// TwinCAT 3 PLC project PLC1
// ProgramVersion: 3.1.4020.5
// libraries:
//   Tc2_ModbusRTU, * (Beckhoff Automation GmbH)
//   Tc2_SerialCom, * (Beckhoff Automation GmbH)
//   Tc2_Standard, * (Beckhoff Automation GmbH)
//   Tc2_System, * (Beckhoff Automation GmbH)
//   Tc3_Module, * (Beckhoff Automation GmbH)
// project tree:
//   DUTs/SH200A/ ST_LoggedValues.TcDUT, ST_Simplex_Halt.TcDUT, ST_Simplex_Jog.TcDUT, ST_Simplex_Reset.TcDUT, ST_Simplex_SetPosition.TcDUT, ST_Simplex_Stop.TcDUT
//   / PlcTask.TcTTO
//   POUs/ FB_Simplex.TcPOU, MAIN.TcPOU
//   POUs/ModbusRTU/ ModbusRTU.TcGVL, SerialCommunication.TcPOU
// real-time tasks:
//   TASK PlcTask: cycle T#2ms, priority 20, ADS port 350
// I/O:
//   DEVICE Device 1 (EtherCAT), AmsNetId 192.168.1.100.2.1
//     Term 1 (EK1200) [EK1200-5000 EtherCAT Power supply (2A E-Bus)]
//       Term 2 (EL1008) [EL1008 8Ch. Dig. Input 24V, 3ms]
//       Term 3 (EL2008) [EL2008 8Ch. Dig. Output 24V, 0.5A]
//       Term 4 (EL9510) [EL9510 Power supply terminal 10V]
//       Term 5 (EL3356) [EL3356 1Ch. Ana. Input Resistor Bridge Terminal, 16bit, High Precision]
//       Term 6 (EL9011) [EL9011 End Terminal]
//   DEVICE Device 3 (EtherCAT), AmsNetId 192.168.1.100.4.1
//     Term 7 (EP6002-0002) [EP6002-0002 Interface (RS232/422/485)]
//   DEVICE Device 2 (COM Port)
// variable links:
//   PLC1/PLC1 Instance <-> Device 3 (EtherCAT)/Term 7 (EP6002-0002)
//     PlcTask Inputs/MAIN.fbSH200A.fbModbusRTUMaster.InData/D <-> COM TxPDO-Map Inputs Channel 1/Data In 0
//     PlcTask Inputs/MAIN.fbSH200A.fbModbusRTUMaster.InData/D @bit {8..168 step 8} <-> COM TxPDO-Map Inputs Channel 1/Data In {1..21}  (21 links)
//     PlcTask Inputs/MAIN.fbSH200A.fbModbusRTUMaster.InData/Status <-> COM TxPDO-Map Inputs Channel 1/Status
//     PlcTask Outputs/MAIN.fbSH200A.fbModbusRTUMaster.OutData/Ctrl <-> COM RxPDO-Map Outputs Channel 1/Ctrl
//     PlcTask Outputs/MAIN.fbSH200A.fbModbusRTUMaster.OutData/D <-> COM RxPDO-Map Outputs Channel 1/Data Out 0
//     PlcTask Outputs/MAIN.fbSH200A.fbModbusRTUMaster.OutData/D @bit {8..168 step 8} <-> COM RxPDO-Map Outputs Channel 1/Data Out {1..21}  (21 links)

CONFIGURATION PLC1
    RESOURCE PLC ON TwinCAT3
        TASK PlcTask(INTERVAL := T#2ms, PRIORITY := 20);
        PROGRAM MAIN WITH PlcTask : MAIN;
    END_RESOURCE
END_CONFIGURATION

// ---- DUTs/SH200A/ST_LoggedValues.TcDUT
TYPE ST_LoggedValues :
STRUCT
	nMotorFluxVoltage : INT;
END_STRUCT
END_TYPE

// ---- DUTs/SH200A/ST_Simplex_Halt.TcDUT
TYPE ST_Simplex_Halt :
STRUCT
	nMotorFluxVoltage : INT;
END_STRUCT
END_TYPE

// ---- DUTs/SH200A/ST_Simplex_Jog.TcDUT
TYPE ST_Simplex_Jog :
STRUCT
	fbTimerWriteModbus		: TON;		// Timer for writing values to Modbus
	bWriteControlOption		: BOOL;		// First state, define control mode
		nControlSetting		: UINT := 21; // Default value is set to position ramp control
	bWriteSetpointSpeed		: BOOL; 	// Second state, define maximum speed
		nMaxVelocity		: INT; 		// Maximum allowed velocity
		bSettingsDone		: BOOL;
	bJogForward				: BOOL;		// Third state, jogging forwards
	bJogBackwards			: BOOL;		// Fourth state, jogging backwards
		fbTimerWritePosition : TON;
		bSendPosition_MSB	: BOOL; // New setpoint sent to the motor Register! 
		bSendPosition_LSB	: BOOL; // New setpoint sent to the motor Register!
		bReadPosition		: BOOL;	// State inside jogg (all data is sent) 
	dnPosition				: DINT; // Current position of the motor
	
	//fAcceleration:LREAL;
	//fDeceleration:LREAL;
	//fJerk:LREAL;
	bDone	: BOOL;
	bBusy	: BOOL;
	bActive	: BOOL;
	bCommandAborted	: BOOL;
	bError	 : BOOL;
	nErrorID : UDINT;
END_STRUCT
END_TYPE

// ---- DUTs/SH200A/ST_Simplex_Reset.TcDUT
TYPE ST_Simplex_Reset :
STRUCT
END_STRUCT
END_TYPE

// ---- DUTs/SH200A/ST_Simplex_SetPosition.TcDUT
TYPE ST_Simplex_SetPosition :
STRUCT
	bExecute:BOOL;
	fPosition:LREAL;
	bMode:BOOL;
	//	stOptions:ST_SetPositionOptions;
	bDone:BOOL;
	bBusy:BOOL;
	bError:BOOL;
	nErrorID:UDINT;
END_STRUCT
END_TYPE

// ---- DUTs/SH200A/ST_Simplex_Stop.TcDUT
TYPE ST_Simplex_Stop :
STRUCT
	bExecute:BOOL;
	fDeceleration:LREAL;
	fJerk:LREAL;
	//stOptions:ST_MoveOptions;
	bDone:BOOL;
	bBusy:BOOL;
	bActive:BOOL;
	bCommandAborted:BOOL;
	bError:BOOL;
	nErrorID:UDINT;
END_STRUCT
END_TYPE

// ---- POUs/ModbusRTU/ModbusRTU.TcGVL
VAR_GLOBAL
	COMin_EL60XX AT %I* : KL6InData22B;
	COMout_EL60XX AT %Q* : KL6OutData22B;
	RxBuffer: Combuffer;
	TxBuffer: Combuffer;
END_VAR

// ---- POUs/MAIN.TcPOU
PROGRAM MAIN
VAR
	fbSH200A : FB_Simplex();
END_VAR

fbSH200A.M_Jog();
//fbSH200A.M_LogValues();
SerialCommunication();
//fbSH200A();

END_PROGRAM

// ---- POUs/FB_Simplex.TcPOU
FUNCTION_BLOCK FB_Simplex
VAR
	(* Stored Motor Parameters *)
	bWriteData	: BOOL;

	nTorqueLimit		: INT  := 3; // TorqueLimit for the motor  
	rM_SetPointSpeed	: REAL := 10;		 // Setpoint from user (cmm/s) 
	unControlOption		: UINT := 32;
	
	dnCenterPosition	: DINT;
	dnCCVEndPosition	: DINT := -200000;
	dnCVEndPosition		: DINT := 200000;

	dnPosRegMSB			: DINT;
	dnPosRegLSB			: DINT;
	
	fbModbusRTUMaster 	: MODbusRtuMaster_KL6x22B;
		unVersionNumber		: UINT;
		bMBAddress			: BYTE;
		unQuantity			: UINT; 
		unMBAddr			: UINT;
		unDataLength		: UINT;
		bStartReading		: BOOL;
		unTimeOut			: TIME := T#5S;	
		bBusy				: BOOL;
		bError				: BOOL;
		unErrorID			: UINT;
		unReadBytes			: UINT;
		lnPosition			: LINT;
		SPosition			: DINT;
		nCurr				: INT; // Read register 223	
	stSimplex_SetPosition	: ST_Simplex_SetPosition();	
	stSimplex_Jog			: ST_Simplex_Jog();
	stSimplex_Stop			: ST_Simplex_Stop();
	stSimplex_Reset			: ST_Simplex_Reset();
	stSimplex_Halt			: ST_Simplex_Halt();
	stLoggedValues			: ST_LoggedValues();
	dnRedMSB: BYTE;
END_VAR

(*		fbModbusRTUMaster(	UnitID   := 1,
						  	Quantity := 2,
							MBAddr	 := 200,
							cbLength := 4,
							pMemoryAddr := ADR(lnPosition),
							Execute		:= bWriteData, 
							TimeOut		:= T#5S, 
							Busy		=> bBusy, 
							Error		=> bError,
							ErrorId		=> unErrorID,
							cbRead		=> unReadBytes);		
		fbModbusRTUMaster.ReadRegs();
 *)
 (*
 	fbModbusRTUMaster(	UnitID   := 1,
					  	Quantity := 1,
						MBAddr	 := 449,
						cbLength := 16,
						pMemoryAddr := ADR(dnPosRegMsb),
						Execute		:= bWriteData, 
						TimeOut		:= T#5S, 
						Busy		=> bBusy, 
						Error		=> bError,
						ErrorId		=> unErrorID,
						cbRead		=> unReadBytes);		
	fbModbusRTUMaster.WriteRegs();
*)

{warning 'add method implementation'}
METHOD M_checkNC_settings : BOOL
VAR_INPUT
	//AXIS_REF	: REFERENCE TO Tc2_MC2.AXIS_REF;
END_VAR
END_METHOD

METHOD M_Jog : BOOL
VAR_INPUT
END_VAR
VAR
	bWrite 	: BOOL;	// Write command to Simplex motor
END_VAR
IF stSimplex_Jog.bActive THEN
	stSimplex_Jog.bWriteControlOption := TRUE;
	stSimplex_Jog.bActive := FALSE;
	stSimplex_Jog.bBusy := TRUE;
END_IF

// State to send setpoint velocity to SH200A
IF stSimplex_Jog.bWriteControlOption THEN
	stSimplex_Jog.fbTimerWriteModbus(PT := T#200MS);
	stSimplex_Jog.fbTimerWriteModbus(IN := TRUE);
	IF stSimplex_Jog.fbTimerWriteModbus.Q THEN
		bWrite := TRUE;
		fbModbusRTUMaster(	UnitID   := 1,
						  	Quantity := 1,
							MBAddr	 := 399,
							cbLength := 2,
							pMemoryAddr := ADR(stSimplex_Jog.nControlSetting),
							Execute		:= bWrite, 
							TimeOut		:= T#5S, 
							Busy		=> bBusy, 
							Error		=> bError,
							ErrorId		=> unErrorID,
							cbRead		=> unReadBytes);		
		stSimplex_Jog.bWriteControlOption := FALSE; 
		stSimplex_Jog.bWriteSetPointSpeed := TRUE;
		stSimplex_Jog.fbTimerWriteModbus(IN := FALSE);
	ELSE
		bWrite := FALSE;
		fbModbusRTUMaster(Execute := FALSE);
	END_IF	
	fbModbusRTUMaster.WriteSingleRegister();
	

// State to send control option to SH200A
ELSIF stSimplex_Jog.bWriteSetpointSpeed THEN 
	IF stSimplex_Jog.bSettingsDone THEN
		stSimplex_Jog.bJogForward 			:= TRUE;
		stSimplex_Jog.bSendPosition_LSB 	:= TRUE; 
		stSimplex_Jog.bSendPosition_MSB 	:= TRUE; 
		stSimplex_Jog.bWriteSetPointSpeed 	:= FALSE;
		stSimplex_Jog.bSettingsDone			:= FALSE;
	END_IF
		
	stSimplex_Jog.fbTimerWriteModbus(PT := T#200MS);
	stSimplex_Jog.fbTimerWriteModbus(IN := TRUE);
	stSimplex_Jog.nMaxVelocity := M_MM_TO_SPEED(rMM_SetPoint := rM_SetPointSpeed);
	
	IF stSimplex_Jog.fbTimerWriteModbus.Q THEN
		bWrite := TRUE;
		fbModbusRTUMaster( UnitID   	:= 1,
						   quantity 	:= 1,
						   MBAddr	 	:= 350,
						   cbLength 	:= 2,
						   pMemoryAddr 	:= ADR(stSimplex_Jog.nMaxVelocity),
						   Execute		:= bWrite, 
						   TimeOut		:= T#5S, 
						   Busy			=> bBusy, 
						   Error		=> bError,
						   ErrorId		=> unErrorID,
						   cbRead		=> unReadBytes);	
		stSimplex_Jog.fbTimerWriteModbus(IN := FALSE);
		stSimplex_Jog.bSettingsDone := TRUE;
	ELSE
		bWrite := FALSE;
		fbModbusRTUMaster(Execute := FALSE);
	END_IF
	fbModbusRTUMaster.WriteSingleRegister();
(* STATE 3: JOGGING FORWARD*)
ELSIF stSimplex_Jog.bJogForward THEN
	// Data formatting for Modbus (protcol is broken in the motor)
	dnPosRegMSB := (dnCVEndPosition AND 2#11111111111111110000000000000000);
	dnPosRegLSB := (dnCVEndPosition AND 2#00000000000000001111111111111111);
	
	// If we are done with set-up of new set point read the position for the motor
	IF stSimplex_Jog.bReadPosition THEN
		// Read position from motor
		bWrite := TRUE;
		fbModbusRTUMaster( 	UnitID   	:= 1,
					  		Quantity 	:= 2,
					   		MBAddr	 	:= 200,
					   		cbLength 	:= 4,
					   		pMemoryAddr := ADR(stSimplex_Jog.dnPosition),
					   		Execute		:= bWrite, 
					   		TimeOut		:= T#5S, 
					   		Busy		=> bBusy, 
					   		Error		=> bError,
					   		ErrorId		=> unErrorID,
					   		cbRead		=> unReadBytes);		
		stSimplex_Jog.fbTimerWriteModbus(IN := FALSE);
		fbModbusRTUMaster.ReadRegs();
		IF NOT(bBusy) AND unReadBytes <> 0 THEN
			bWrite := FALSE;
			fbModbusRTUMaster.Execute := FALSE;
		END_IF
	END_IF
	
	IF stSimplex_Jog.bSendPosition_LSB AND stSimplex_Jog.bSendPosition_MSB THEN
		stSimplex_Jog.fbTimerWriteModbus(PT := T#10MS);
		stSimplex_Jog.fbTimerWriteModbus(IN := TRUE);
		
		IF stSimplex_Jog.fbTimerWriteModbus.Q THEN
			fbModbusRTUMaster(	UnitID   := 1,
								Quantity := 1,
								MBAddr	 := 449,
								cbLength := 16,
								pMemoryAddr := ADR(dnPosRegMSB),
								Execute		:= bWrite, 
								TimeOut		:= T#5S, 
								Busy		=> bBusy, 
								Error		=> bError,
								ErrorId		=> unErrorID,
								cbRead		=> unReadBytes);		
			fbModbusRTUMaster.WriteRegs();
			StSimplex_Jog.bSendPosition_MSB := FALSE;
			stSimplex_Jog.fbTimerWriteModbus(IN := FALSE);
		ELSE
			bWrite := FALSE;
			fbModbusRTUMaster(Execute := FALSE);
		END_IF
	ELSIF NOT(stSimplex_Jog.bSendPosition_MSB) AND stSimplex_Jog.bSendPosition_LSB THEN
		stSimplex_Jog.fbTimerWriteModbus(PT := T#10MS);
		stSimplex_Jog.fbTimerWriteModbus(IN := TRUE);
		
		IF stSimplex_Jog.fbTimerWriteModbus.Q THEN
			bWrite := TRUE;
			fbModbusRTUMaster(	UnitID   := 1,
								Quantity := 1,
								MBAddr	 := 450,
								cbLength := 16,
								pMemoryAddr := ADR(dnPosRegLSB),
								Execute		:= bWrite, 
								TimeOut		:= T#5S, 
								Busy		=> bBusy, 
								Error		=> bError,
								ErrorId		=> unErrorID,
								cbRead		=> unReadBytes);		
			fbModbusRTUMaster.WriteRegs();
			StSimplex_Jog.bSendPosition_LSB := FALSE;	
			stSimplex_Jog.fbTimerWriteModbus(IN := FALSE);
		ELSE
			bWrite := FALSE;
			fbModbusRTUMaster(Execute := FALSE);
		END_IF
	ELSIF NOT(stSimplex_Jog.bSendPosition_MSB) AND NOT(stSimplex_Jog.bSendPosition_LSB) THEN
		fbModbusRTUMaster.WriteRegs();
		stSimplex_Jog.bReadPosition := TRUE;
	END_IF		

	IF stSimplex_Jog.dnPosition >= dnCVEndPosition THEN
		stSimplex_Jog.bJogForward		:= FALSE;
		stSimplex_Jog.bJogBackwards 	:= TRUE;
		stSimplex_Jog.bReadPosition 	:= FALSE;
		stSimplex_Jog.bSendPosition_LSB := TRUE;
		stSimplex_Jog.bSendPosition_MSB := TRUE;
		fbModbusRTUMaster.Execute 		:= FALSE;
	END_IF

(* STATE 4: JOGGING BACKWARDS*)
ELSIF stSimplex_Jog.bJogBackwards THEN
	dnPosRegMSB := (dnCCVEndPosition AND 2#11111111111111110000000000000000);
	dnPosRegLSB := (dnCCVEndPosition AND 2#00000000000000001111111111111111);
	
	// Read the position of the motor (True if we are done with the set-up)
	IF stSimplex_Jog.bReadPosition THEN
		// Read position from motor
		bWrite := TRUE;
		fbModbusRTUMaster( 	UnitID   	:= 1,
					  		Quantity 	:= 2,
					   		MBAddr	 	:= 200,
					   		cbLength 	:= 4,
					   		pMemoryAddr := ADR(stSimplex_Jog.dnPosition),
					   		Execute		:= bWrite, 
					   		TimeOut		:= T#5S, 
					   		Busy		=> bBusy, 
					   		Error		=> bError,
					   		ErrorId		=> unErrorID,
					   		cbRead		=> unReadBytes);		
		fbModbusRTUMaster.ReadRegs();
		IF NOT(bBusy) AND unReadBytes <> 0 THEN
			bWrite := FALSE;
			fbModbusRTUMaster.Execute := FALSE;
		END_IF
	END_IF		
	
	IF stSimplex_Jog.bSendPosition_LSB AND stSimplex_Jog.bSendPosition_MSB THEN
		stSimplex_Jog.fbTimerWriteModbus(PT := T#10MS);
		stSimplex_Jog.fbTimerWriteModbus(IN := TRUE);
		
		IF stSimplex_Jog.fbTimerWriteModbus.Q THEN
			fbModbusRTUMaster(	UnitID   := 1,
								Quantity := 1,
								MBAddr	 := 449,
								cbLength := 16,
								pMemoryAddr := ADR(dnPosRegMSB),
								Execute		:= bWrite, 
								TimeOut		:= T#5S, 
								Busy		=> bBusy, 
								Error		=> bError,
								ErrorId		=> unErrorID,
								cbRead		=> unReadBytes);
			stSimplex_Jog.fbTimerWriteModbus(IN := FALSE);
			fbModbusRTUMaster.WriteRegs();
			StSimplex_Jog.bSendPosition_MSB := FALSE;
		ELSE
			bWrite := FALSE;
			fbModbusRTUMaster(Execute := FALSE);
		END_IF
	ELSIF NOT(stSimplex_Jog.bSendPosition_MSB) AND stSimplex_Jog.bSendPosition_LSB THEN	
		stSimplex_Jog.fbTimerWriteModbus(PT := T#10MS);
		stSimplex_Jog.fbTimerWriteModbus(IN := TRUE);
		
		IF stSimplex_Jog.fbTimerWriteModbus.Q THEN
			bWrite := TRUE;
			fbModbusRTUMaster(	UnitID   := 1,
								Quantity := 1,
								MBAddr	 := 450,
								cbLength := 16,
								pMemoryAddr := ADR(dnPosRegLSB),
								Execute		:= bWrite, 
								TimeOut		:= T#5S, 
								Busy		=> bBusy, 
								Error		=> bError,
								ErrorId		=> unErrorID,
								cbRead		=> unReadBytes);
			stSimplex_Jog.fbTimerWriteModbus(IN := FALSE);		
			fbModbusRTUMaster.WriteRegs();
			StSimplex_Jog.bSendPosition_LSB := FALSE;	
		ELSE
			bWrite := FALSE;
			fbModbusRTUMaster(Execute := FALSE);
		END_IF
	ELSIF NOT(stSimplex_Jog.bSendPosition_MSB) AND NOT(stSimplex_Jog.bSendPosition_LSB) THEN
		fbModbusRTUMaster.WriteRegs();
		stSimplex_Jog.bReadPosition := TRUE;
	END_IF
	
	IF stSimplex_Jog.dnPosition >= dnCCVEndPosition THEN
		stSimplex_Jog.bJogForward		:= TRUE;
		stSimplex_Jog.bJogBackwards 	:= FALSE;
		stSimplex_Jog.bReadPosition 	:= FALSE;
		stSimplex_Jog.bSendPosition_LSB := TRUE;
		stSimplex_Jog.bSendPosition_MSB := TRUE;
		fbModbusRTUMaster.Execute 		:= FALSE;
	END_IF	
END_IF

IF stSimplex_Jog.bDone OR stSimplex_Jog.bCommandAborted THEN
	stSimplex_Jog.bJogForward			:= FALSE;
	stSimplex_Jog.bJogBackwards 		:= FALSE;
	stSimplex_Jog.bWriteSetpointSpeed 	:= FALSE;
	stSimplex_Jog.bWriteControlOption 	:= FALSE;
	stSimplex_Jog.bBusy   				:= FALSE;
	stSimplex_Jog.bActive 				:= FALSE;
END_IF
END_METHOD

METHOD M_LogValues : BOOL
VAR_INPUT
	//AXIS_REF	: REFERENCE TO Tc2_MC2.AXIS_REF;
END_VAR
VAR
	nValue : INT;
	nReadBytes : UINT;
END_VAR
(*
IF NOT(bBusy) THEN
	fbModbusRTUMaster(	UnitID   := 1,
					  	Quantity := 1,
						MBAddr	 := 208,
						cbLength := 2,
						pMemoryAddr := ADR(nValue),
						Execute		:= TRUE, 
						TimeOut		:= T#5S, 
						Busy		=> bBusy, 
						Error		=> bError,
						ErrorId		=> unErrorID,
						cbRead		=> nReadBytes);		
	fbModbusRTUMaster.WriteSingleRegister();
END_IF
IF nReadBytes <> 0 THEN
	stLoggedValues.nMotorFluxVoltage := nValue;
END_IF
*)
// Typiskt är 50/200 mm per varv = 0.25 mm per varv 

// 400, uint, värde 32 är speed control för position (Håll en viss fart till position är uppnått) 




// 340, int, unit is positions per second / 16, 0..25600
END_METHOD

METHOD M_MM_TO_SPEED : INT;
VAR_INPUT
	rMM_SetPoint : REAL; 
END_VAR
M_MM_TO_SPEED := REAL_TO_INT(rMM_Setpoint*256*0.25);
END_METHOD

{warning 'add method implementation'}
METHOD M_ResetDrive : BOOL
VAR_INPUT
	//AXIS_REF	: REFERENCE TO Tc2_MC2.AXIS_REF;
END_VAR
END_METHOD

{warning 'add method implementation'}
METHOD M_SetPositionOffset : BOOL
VAR_INPUT
	//AXIS_REF	: REFERENCE TO Tc2_MC2.AXIS_REF;
END_VAR
VAR
	//stMC_SetPosition : ST_MC_SetPosition;
END_VAR
VAR CONSTANT
	// Variables for calculation of the speed
END_VAR
//stMC_Setposition.bExecute := TRUE;
END_METHOD

METHOD M_SetSpeed : BOOL
VAR_INPUT
	//AXIS_REF	: REFERENCE TO Tc2_MC2.AXIS_REF;
END_VAR
VAR
	bState1 	: BOOL; // Write setpoint
	bState2		: BOOL; // Start moving 
	bState3		: BOOL; // Error or end position reach 
END_VAR
// Typiskt är 50/200 mm per varv = 0.25 mm per varv 

// 400, uint, värde 32 är speed control för position (Håll en viss fart till position är uppnått) 




// 340, int, unit is positions per second / 16, 0..25600
END_METHOD

{warning 'add method implementation'}
METHOD M_SetTorqueLimit : BOOL
VAR_INPUT
	//AXIS_REF	: REFERENCE TO Tc2_MC2.AXIS_REF;
END_VAR
VAR_OUTPUT
	bQued	: BOOL;	
END_VAR
VAR
	bBusy 		: BOOL;
	bExecute	: BOOL;
	bError		: BOOL;
	unErrorID	: UINT; 
	nReadBytes	: UINT;
END_VAR
(*// Write register 203!! 
fbModbusRTUMaster(	UnitID   := 1,
				  	Quantity := 1,
					MBAddr	 := 204,
					cbLength := 1,
					pMemoryAddr := ADR(nTorqueLimit),
					Execute		:= TRUE, 
					TimeOut		:= T#5S, 
					Busy		=> bBusy, 
					Error		=> bError,
					ErrorId		=> unErrorID,
					cbRead		=> nReadBytes);
				

IF NOT(bBusy) THEN
	fbModbusRTUMaster.WriteSingleRegister();
	bQued	:= FALSE;
ELSE
	bQued	:= TRUE;
END_IF
*)
END_METHOD

METHOD M_SetZeroRef : BOOL
VAR_INPUT
END_VAR
END_METHOD

END_FUNCTION_BLOCK

// ---- POUs/ModbusRTU/SerialCommunication.TcPOU
PROGRAM SerialCommunication
VAR
	COMportControl: SerialLineControl;
	COMportControlError: BOOL;
	COMportControlErrorID: ComError_t;
END_VAR

(*==================================================================
	Background communication with KL6001 terminal
	The SerialLineControl function block is supposed to be called in every PLC cycle.
	It communicates with the serial line hardware device and transmits or receives data.
	The SerialLineControl can be called in the standard task or in a separate fast task as well.
	A fast separate task will be necessary at high baud rates or 
	with KL6001 terminals which have a small process image (3 or 5 data bytes only)
*)
COMportControl(
	Mode:= SERIALLINEMODE_EL6_22B,
	pComIn:= ADR(COMin_EL60xx),			(* I/O data; see global variables *)
	pComOut:= ADR(COMout_EL60xx),		(* I/O data; see global variables *)
	SizeComIn:= SIZEOF(COMin_EL60xx),	(* I/O data; see global variables *)
	TxBuffer:= TxBuffer,				(* transmit buffer; see global variables *)
	RxBuffer:= RxBuffer,				(* receive buffer; see global variables *)
	Error=> COMportControlError,
	ErrorID=> COMportControlErrorID );

END_PROGRAM
